{attribute 'linkalways'} 
{attribute 'no_explicit_call' := 'This FB is a CLASS and must be accessed using methods or properties'}
{attribute 'enable_dynamic_creation'}
FUNCTION_BLOCK FINAL AND_USINT EXTENDS Node
VAR
	in1 : _USINT(0);
	in2 : _USINT(0);
	out : _USINT(0);
END_VAR

METHOD PUBLIC Clone : I_Node
VAR
	pNode : POINTER TO AND_USINT;
END_VAR
pNode := __NEW(AND_USINT);
Clone := pNode^;
END_METHOD

METHOD FB_init : BOOL
VAR_INPUT
	bInitRetains : BOOL; // if TRUE, the retain variables are initialized (warm start / cold start)
	bInCopyCode : BOOL;  // if TRUE, the instance afterwards gets moved into the copy code (online change)
END_VAR
AddInput('in1',THIS^.in1);
AddInput('in2',THIS^.in2);
AddOutput('out', THIS^.out);
END_METHOD

METHOD PROTECTED OnExecute
VAR
END_VAR
out.Value := in1.Value AND in2.Value;
END_METHOD

END_FUNCTION_BLOCK

(* stored: Version 1.1.0.1, ProductVersion 3.1.4024.15
   POU AND_USINT: Id {319d0d26-e920-497c-a2fb-51a935a3f0b0}, SpecialFunc None
   Folder Constructor: Id {a01dc9f5-b4a6-4425-ac94-3315ff91a1bb}
   Method Clone: Id {48da2861-ef3d-4966-885f-1cab22456a33}
   Method FB_init: Id {55c73731-a95f-4438-8af8-ac0414df4949}
   Method OnExecute: Id {6e55ee1b-96e3-482e-b5e5-b144a794c6f5} *)
